// TIA Portal V20 export
DATA_BLOCK "DB_PrioSequence"   // DB114
// stored: InstanceOfName FB_PrioSequence, InstanceOfType FB
"FB_PrioSequence"
   // VAR
   //    sPrio : Int;
   // END_VAR
BEGIN
END_DATA_BLOCK
